(* CoDeSys 2.3 export: TRANSFER_AIR.EXP *)

(* POU Transfer_Air, ST *)
FUNCTION Transfer_Air : BYTE
VAR_INPUT
	IN: INT;				(* input value*)
END_VAR
VAR
	IN_MIN:REAL := 0;			(* minimum input value *)
	IN_MAX:REAL := 100;			(* maximum input value *)
	OUT_MIN:REAL := 0;		(* corresponding minimum output value *)
	OUT_MAX:REAL  := 255;		(* corresponding maximum output value *)
	Diff: REAL;
END_VAR
	Diff := IN_MAX-IN_MIN;
	Transfer_Air :=REAL_TO_BYTE((IN-IN_MIN)/Diff * (OUT_MAX-OUT_MIN) + OUT_MIN);
END_FUNCTION
